// Mitsubishi GX Works2 project: 240507_timechart11_한번on두번off   PLC: Q03UDV

PROGRAM MAIN
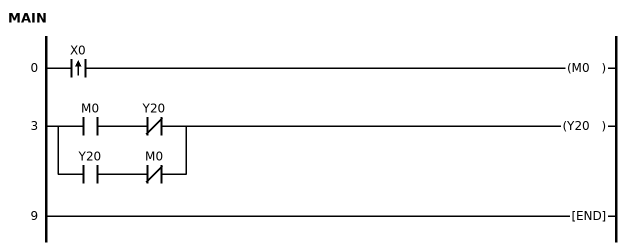
0     LDP     X0
      OUT     M0
3     LD      M0
      ANI     Y20
      LD      Y20
      ANI     M0
      ORB
      OUT     Y20
9     END
END_PROGRAM
